// SIMATIC S7-200 SMART project (STEP 7-Micro/WIN SMART), CPU SR40

ORGANIZATION_BLOCK MAIN:OB1
TITLE=程序注释
BEGIN
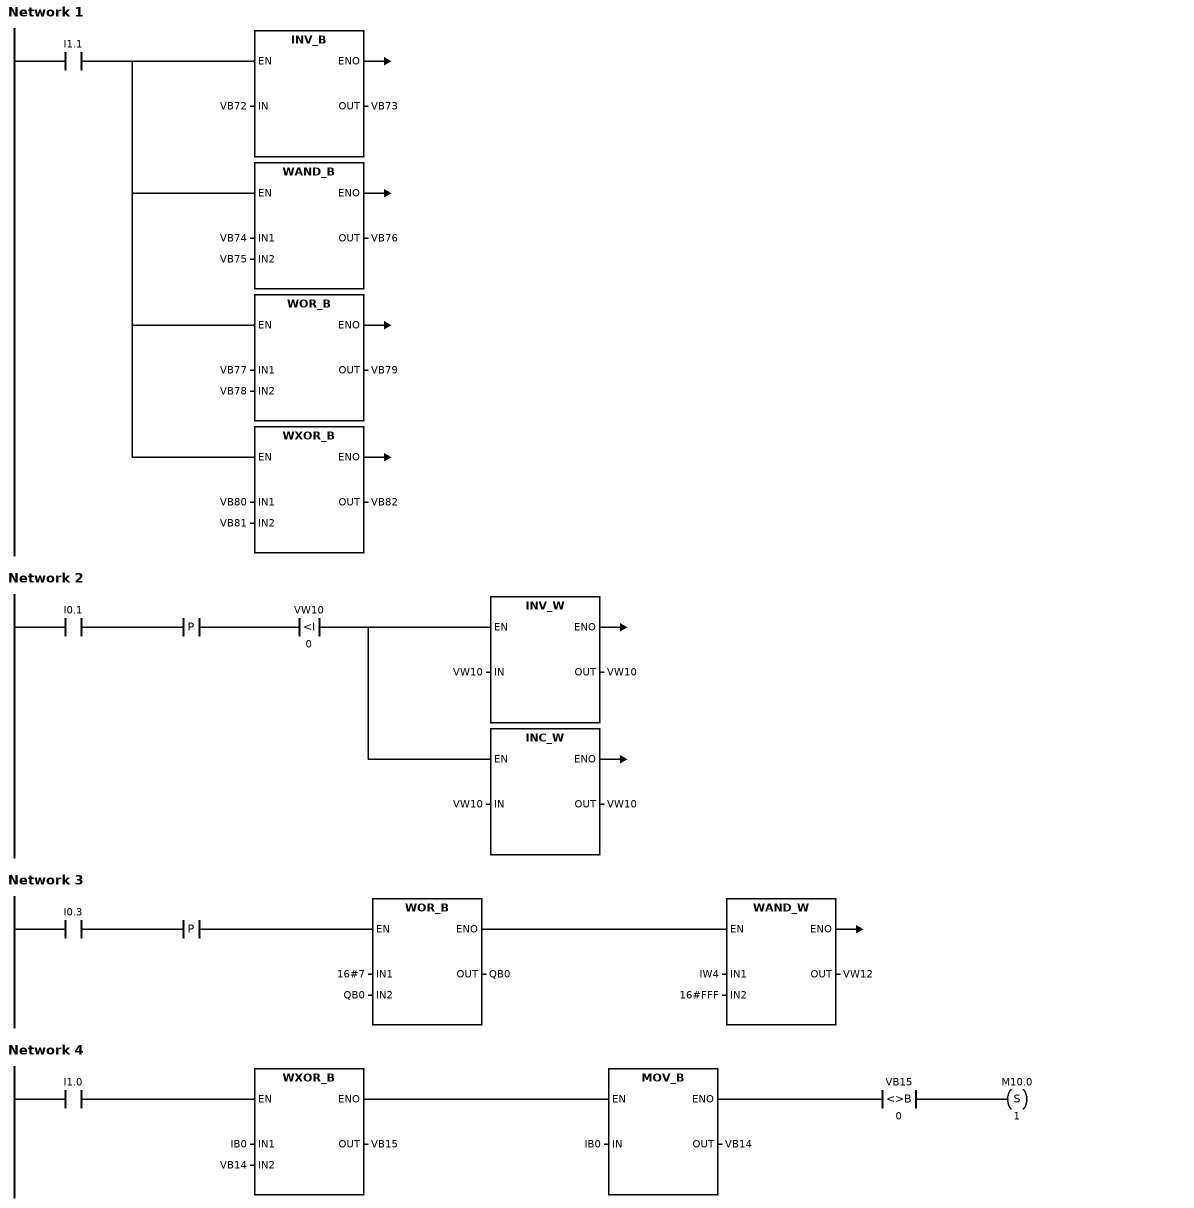
Network 1
LD     I1.1
MOVB   VB72, VB73
INVB   VB73
MOVB   VB74, VB76
ANDB   VB75, VB76
MOVB   VB77, VB79
ORB    VB78, VB79
MOVB   VB80, VB82
XORB   VB81, VB82
Network 2
LD     I0.1
EU
AW<    VW10, 0
INVW   VW10
INCW   VW10
Network 3
LD     I0.3
EU
ORB    16#7, QB0
AENO
MOVW   IW4, VW12
ANDW   16#FFF, VW12
Network 4
LD     I1.0
MOVB   IB0, VB15
AENO
XORB   VB14, VB15
AENO
MOVB   IB0, VB14
AENO
AB<>   VB15, 0
S      M10.0, 1
Network 5
// 程序段注释
END_ORGANIZATION_BLOCK
